(* PLC project BlogProject.project, CODESYS CODESYS V3.5 SP14 Patch 3 *)
(* stored: creationDateTime 2021-10-07T21:05:11.7902533, modificationDateTime 2021-10-07T20:40:20.1109198 *)

FUNCTION_BLOCK mcIsSystemChecked IMPLEMENTS itfEvent
  VAR
    bSystemCheck : BOOL;
  END_VAR

            
          

METHOD getEvent : BOOL
                  getEvent:=bSystemCheck;
                
END_METHOD
END_FUNCTION_BLOCK
